FUNCTION_BLOCK FB_TRK_BASE EXTENDS FB_MA_BASE
VAR_INPUT
END_VAR
VAR_OUTPUT
END_VAR
VAR
	{attribute 'OPC.UA.DA' := '0'}
	TrkCfg:		        REFERENCE TO T_TRK_CFG;	    // Reference to Config parameters
	{attribute 'OPC.UA.DA' := '0'}
	TrkCtrl:		    REFERENCE TO T_TRK_CTRL;	// Reference to Control parameters
	{attribute 'OPC.UA.DA' := '0'}
	TrkStat:		    REFERENCE TO T_TRK_STAT;	// Reference to Status parameters
	
    // Tracking data structure (TrackingData) is defined in C++ module
	{attribute 'OPC.UA.DA' := '0'}
	i_trk_data          AT %I*: PointingKernelPositions;
	
	{attribute 'OPC.UA.DA' := '0'}
	i_ccs_data          AT %I*: CcsData;
	
	
	
END_VAR



SUPER^();

// Method for hard-coding of configuration parameters by the User.
METHOD User_Configure : BOOL
VAR_INPUT
END_VAR
VAR
	i:	INT;
END_VAR
SUPER^.User_Configure();	// Mandatory!
END_METHOD

// User Method executed on each cycle before processing events and states.
METHOD User_GetParams : BOOL
VAR_INPUT
END_VAR
VAR
	i:	INT;
END_VAR

// Assign output variables according input configuration and control.
END_METHOD

// User Method executed on each cycle after processing events and states.
METHOD User_SetParams : BOOL
VAR_INPUT
END_VAR
VAR
	i:		INT;
END_VAR

memcpy(ADR(TrkCfg.site), ADR(i_ccs_data.site), SIZEOF(TrkCfg.site));
memcpy(ADR(TrkCtrl.environment), ADR(i_ccs_data.environment), SIZEOF(TrkCtrl.environment));
memcpy(ADR(TrkStat.data), ADR(i_trk_data), SIZEOF(TrkStat.data));
memcpy(ADR(TrkStat.data_deg), ADR(i_trk_data), SIZEOF(TrkStat.data_deg));
TrkStat.data_deg.target_observed_altaz[0] := RAD_TO_DEG(TrkStat.data.target_observed_altaz[0]);
TrkStat.data_deg.target_observed_altaz[1] := RAD_TO_DEG(TrkStat.data.target_observed_altaz[1]);
TrkStat.data_deg.parallactic_angle := RAD_TO_DEG(TrkStat.data.parallactic_angle);
TrkStat.data_deg.north_angle := RAD_TO_DEG(TrkStat.data.north_angle);
TrkStat.data_deg.pupil_angle := RAD_TO_DEG(TrkStat.data.pupil_angle);
TrkStat.apparent.alpha := F_astroRad2Hms(i_trk_data.radec_at_altaz_at_requested_xy[0]);
TrkStat.apparent.delta := F_astroRad2Dms(i_trk_data.radec_at_altaz_at_requested_xy[1]);
END_METHOD

END_FUNCTION_BLOCK

(* stored: Version 1.1.0.1, ProductVersion 3.1.4024.10
   POU FB_TRK_BASE: Id {d871ca53-874f-42bb-88fc-5db6d0c7481a}, SpecialFunc None
   Method User_Configure: Id {9b18327f-ebf5-4feb-8255-0ce66dcb8b1c}
   Method User_GetParams: Id {63c9401f-847d-4168-b01e-0e9a29ae6907}
   Method User_SetParams: Id {4e55ee67-727b-4702-b0e3-c4bec93cdfee} *)
